(* CoDeSys 2.3.9.47 project: mqmod.pro *)
(* Libraries: C:\Program Files\WAGO Software\CoDeSys V2.3\Targets\WAGO\Libraries\32_Bit\oscat_basic_333.lib 9.2.16 18:15:54, WagoLibModbus_IP_01.lib 11.2.16 18:05:40, SysLibSockets.lib 22.5.14 16:16:32, WagoLibEthernet_01.lib 11.2.16 18:05:44, Standard.lib 20.5.14 08:13:26, Iecsfc.lib 16.5.13 14:00:50, SYSLIBCALLBACK.LIB 16.5.13 14:00:50 *)

(* PLC configuration (modules and I/O channels)
K-Bus [K_Bus] node 0, in %IB0 out %QB0 {KbusBusMode = 1; KbusCycleTime = 10000; KbusThreadPriority = 0; KbusSetOutputsToZeroOnApplicationStop = 1}
Modbus variables [PFC200MODBUS] node 1, in %IB0 out %QB0 {PlcStopBehaviour = 1; FiledbusErrorBehaviour = 1; TcpOperation = 1; TcpPort = 502; TcpTimeout = 600; UdpOperation = 1; UdpPort = 502; RtuOperation = 0; NodeId = 1; ResponseTimeout = 5000; Interface = 0; Baud = 115200; StopBits = 1; Parity = 1; FlowCtrl = 0; PhysInterface = 0}
Modbus-Master [MB_MASTER] node 2, in %IB0 out %QB0
*)

(* Global variable list: Globale_Variablen *)
VAR_GLOBAL
	xxSubscribe: BOOL := TRUE;
	xxPublish : BOOL     := TRUE;
	SubPubState : INT;
END_VAR

(* Data type *)
TYPE Buffer :
STRUCT
	data : ARRAY [0..MAX_RECEIVE_TCP_CLIENT] OF BYTE;
	iPos : DWORD := 0;
END_STRUCT
END_TYPE

(* Data type *)
TYPE ConnectFlags :
STRUCT
	xUsername     : BOOL;
	xPassword     : BOOL;
	xWillRetain   : BOOL;
	xWillQoS1     : BOOL;
    xWillQoS2     : BOOL;
	xWillFlag     : BOOL;
	xCleanSession : BOOL;
END_STRUCT
END_TYPE

(* Data type *)
TYPE FixedHeader :
STRUCT
	bMessageType : BYTE := 16#00;
	xDUP_FLAG    : BOOL := FALSE;
	xQos         : BYTE := 16#00; (*0,1,2*)
	xRetain      : BOOL := FALSE;
END_STRUCT
END_TYPE

(* Data type *)
TYPE FixedHeaderSub :
STRUCT
	bMessageType : BYTE := 8;
	xReserved         : BYTE := 2;
END_STRUCT
END_TYPE

(* Data type *)
TYPE Payload :
STRUCT
	data : ARRAY [0..30] OF BYTE;
	iPos : DWORD := 0;
END_STRUCT
END_TYPE

(* Data type *)
TYPE typReadReq :
STRUCT
	xReadRegister				:BOOL;
	wAdrBlockStart				:WORD;
	wAdrBlockQuantity			:WORD;
	ptDATA					:POINTER TO BYTE;
END_STRUCT
END_TYPE

(* Data type *)
TYPE typWriteReq
STRUCT
	xWriteRegister				:BOOL;
	wAdrBlockStart				:WORD;
	wAdrBlockQuantity			:WORD;
	ptDATA					:POINTER TO BYTE;
END_STRUCT
END_TYPE

(* POU PLC_PRG, ST *)
PROGRAM PLC_PRG
VAR

(*MQTT COMMUNICATION*)
	mqttClient: MQTT_CLIENT;
	xPublish: BOOL;
	xSubscribe: BOOL;
	socModbus : MODBUS_MASTER;

END_VAR
mqttClient(
xPublish := xxPublish, (* I/O variable to publish to a TOPIC *)
xSubscribe := xxSubscribe,  (* NOT SUPPORTED, but must be here for I/O *)
sIP:='10.210.10.29', (* IP of the MQTT Broker *)
wPortNumber:=1883,  (* PORT of the MQTT Broker *)
(* AUTH: When no authentication is needed, leave the following fields Blank *)
sUsername:='',  (* Username to connect with the MQTT Broker *)
sPassword:='' (* password to connect with the MQTT Broker *)
);

mqttClient.sTopic[1] 	:= 'si/upperstate'; 	(*40705 *)
mqttClient.sTopic[2] 	:= 'si/lowerstate';  	(*40707 *)
mqttClient.sTopic[3] 	:= 'si/activepower';	(*40149*)
mqttClient.sTopic[4]		:= 'si/activate';		(*40151*)
mqttClient.sTopic[5]		:= 'si/deactivate';	(*40151*)

mqttClient.sQoS := 16#00;
mqttClient.pTopic := 'soc';
mqttClient.pQoS := 16#00;
mqttClient.pRetained := FALSE;
mqttClient.pPayload :=  WORD_TO_STRING(socModbus.awRead[2]);(*STRING_TO_UDINT(g_SOC)*);

socModbus(
	xCONNECT:= TRUE,
	strIP_ADDRESS:= '10.210.10.63',
	wPORT:= 502,
	bUNIT_ID:= 16#03,
	bFUNCTION_CODE:= 16#03,
	wREAD_ADDRESS:= 30845 ,
	wREAD_QUANTITY:= 2 ,
 );
END_PROGRAM

(* POU MQTT/MQTT_CLIENT, ST *)
FUNCTION_BLOCK MQTT_CLIENT
VAR CONSTANT
	VERSION 	: BYTE := 16#03;
	Reserved   	: BYTE := 0;
	CONNECT     : BYTE := 1;
	CONNACK     : BYTE := 2;
	PUBLISH     : BYTE := 3;
	PUBACK      : BYTE := 4;
	PUBREC      : BYTE := 5;
	PUBREL      : BYTE := 6;
	PUBCOMP     : BYTE := 7;
	SUBSCRIBE   : BYTE := 8;
	SUBACK      : BYTE := 9;
	UNSUBSCRIBE : BYTE := 10;
	UNSUBACK    : BYTE := 11;
	PINGREQ     : BYTE := 12;
	PINGRESP    : BYTE := 13;
	DISCONNECT  : BYTE := 14;
	Reserved2   : BYTE := 15;

	CONNECTED   : INT := 30;
	NOT_CONNECTED: INT := 40;
	TIMEOUT : INT := 50;
	WAIT_RESPONSE : INT := 60;

	CONNECTION_TIMEOUT : TIME := t#10s;

	SUBSCRIBED : INT := 70;
	PUBLISHED : INT := 80;
	WAIT_RESPONSE_PUBLISH : INT := 90;
END_VAR

VAR
	fixedHeaderSub : BYTE;
	sendBuffer : Buffer;
	receiveBuffer : Buffer;
	fixedHeader: FixedHeader;
	variableHeader: Buffer;
	payLoad:  Buffer;
	connectFlags: ConnectFlags;
	tcpClient: TCP_Client;
	xTcpConnected: BOOL := FALSE;
	xStartSend: BOOL := FALSE;
	diReceiveCount: DINT;
	connectionTimer: TON;
	xTimeOut: BOOL;
	incomingMessageType: BYTE;
	eState: INT;
	xStartTimer: BOOL;

	rawdata : Buffer;
	b : Buffer;
	i :  DINT := 0;
	j:   DINT;
	x:  INT;
	z : INT := 0;

	c : BOOL; (*control state of subscription*)

	modControlValue : ARRAY[0..30] OF BYTE;
	RM : INT;
	LSB : INT;
	modValue : DINT;
	writeAdr : WORD;
	sstopic : ARRAY[0..20] OF BYTE;
	t : STRING;

	modbusMaster : MODBUS_MASTER;

END_VAR

VAR_INPUT
	sTopic: ARRAY[1..5] OF STRING;			(*SUB_TOPICS*)
	pTopic: STRING;						(*PUB_TOPICS*)
	pPayload: STRING;
	pRetained : BOOL;
	pQoS : BYTE;
	sQoS : BYTE;							(*von SMA ENERGY METER*)
	sIp : STRING;
	wPortNumber : WORD;
	sUsername : STRING;
	sPassword : STRING;
END_VAR

VAR_IN_OUT
	xPublish: BOOL;
	xSubscribe: BOOL;
END_VAR


VAR_OUTPUT
	xConnected : BOOL := FALSE;
	xBusy : BOOL := FALSE;
	activePowerVal : REAL;
END_VAR
tcpClient.sIPaddress := sIp;
tcpClient.wPortNumber := wPortNumber;

tcpClient.ptSendData := ADR(sendBuffer.data);
tcpClient.diSendCount := sendBuffer.iPos;

tcpClient(xOpenConnection:=TRUE,
xStartSend:=xStartSend,
aReceiveBuffer := receiveBuffer.data,
diReceiveCount := diReceiveCount);

xTcpConnected := tcpClient.xConnected;
xBusy := xStartSend;

IF NOT xTcpConnected THEN
	eState := NOT_CONNECTED;
	xConnected := FALSE;
 	RETURN;
END_IF;

(* INIT *)
payLoad.iPos := 0;
variableHeader.iPos := 0;

connectionTimer(IN:=xStartTimer, PT:=CONNECTION_TIMEOUT-t#2s);
xTimeOut := connectionTimer.Q;

(* Calculate the current state *)
IF xTimeOut THEN
	eState := TIMEOUT;
ELSIF eState <> CONNECTED AND eState <> TIMEOUT AND eState <> WAIT_RESPONSE THEN
	eState := NOT_CONNECTED;
END_IF

(* Execute current state *)
CASE eState OF

CONNECTED:
	IF diReceiveCount <> 0 THEN
		incomingMessageType := receiveBuffer.data[0];
		IF incomingMessageType = SHL(PINGRESP, 4) THEN
			xStartTimer := TRUE;
		END_IF
		IF incomingMessageType = SHL(PUBLISH, 4)  THEN
			_ARRAY_INIT(ADR(rawdata), SIZEOF(rawdata), 0);
			FOR i:=0 TO diReceiveCount-1 BY 1 DO
				rawdata.data[i] := receiveBuffer.data[i];
			END_FOR

			(*extract zuerst topic then payload*)
			RM := rawdata.data[1];
			LSB := rawdata.data[3];
			_ARRAY_INIT(ADR(sstopic), SIZEOF(sstopic), 0);
			i := 0; z := 0;
			FOR z := 4 TO LSB+3 DO
				sstopic[i]	:= rawdata.data[z];
				i := i + 1;
			END_FOR
			t := CONVERT_TO_STRING(sstopic);
			IF STRING_COMPARE(t, 'si/activepower') THEN
				writeAdr := 40149;
			ELSIF STRING_COMPARE(t, 'si/upperstate') THEN
				writeAdr := 40705;
			ELSIF STRING_COMPARE(t, 'si/lowerstate') THEN
				writeAdr := 40707;
			ELSIF STRING_COMPARE(t, 'si/activate') THEN
				writeAdr := 40151;
			ELSIF STRING_COMPARE(t, 'si/deactivate') THEN
				writeAdr := 40151;
			END_IF

			_ARRAY_INIT(ADR(modControlValue), SIZEOF(modControlValue), 0);
			i := 0; z := 0;
			FOR z := LSB+4 TO RM+1  DO
				modControlValue[i] := rawdata.data[z];
				i := i + 1;
			END_FOR
			modValue := REAL_TO_DINT(CONVERT_TO_REAL(modControlValue));
			z := 0;i := 0;
			modbusMaster(
				xCONNECT:= TRUE,
				strIP_ADDRESS:= '10.210.10.63',
				wPORT:= 502,
				bUNIT_ID:= 16#03,
				bFUNCTION_CODE:= 16#10,
				wWRITE_ADDRESS:= writeAdr, (*unterscheiden nach topic*)
				wWRITE_QUANTITY:= 2,
				value:= modValue);

			(*FOR z := 0 TO 15 BY 1 DO
				pValuesPrev[z] := pValues[z];
			END_FOR
			pValuePrev := CONVERT_TO_REAL(pValuesPrev);*)

			(*(*extract timestamp*)
			i := 0;
			FOR x := 13 TO 31 BY 1 DO
				IF x <> 17 AND x <> 20 AND x <> 23 AND x <> 26 AND x <> 29 THEN
						timestampPayload[i] := a.data[x];
					i := i + 1;
				END_IF
			END_FOR
			timestamp := EXTRACT_TIMESTAMP_FROM_PAYLOAD(timestampPayload);*)


		END_IF

		(*FURTHER QoS > 0*)
		IF incomingMessageType = SHL(PUBACK, 4)  THEN
			_ARRAY_INIT(ADR(b), SIZEOF(b), 0);
			FOR i:=0 TO diReceiveCount-1 BY 1 DO
				b.data[i] := receiveBuffer.data[i];
			END_FOR
		END_IF

		diReceiveCount := 0;
	END_IF

	c := xxPublish AND xxSubscribe;
	IF   c   THEN
		SubPubState := SUBSCRIBED;
	ELSE
		SubPubState := PUBLISHED;
	END_IF;

	CASE SubPubState OF
			SUBSCRIBED:
				IF xxSubscribe THEN
					_BUFFER_CLEAR(ADR(sendBuffer), SIZEOF(sendBuffer));

					fixedHeaderSub :=  BYTE_OF_BIT(FALSE, TRUE, FALSE, FALSE, FALSE, FALSE, FALSE, TRUE); (*FIXED_HEADER*)
					(*fixedHeaderSub.bMessageType := SUBSCRIBE;*)

					_BUFFER_PUSH(ADR(variableHeader), 16#00);(* Message ID *)
					_BUFFER_PUSH(ADR(variableHeader), 16#00);

					_BUFFER_PUSH_STRING(ADR(payLoad), sTopic[1] , TRUE);
					_BUFFER_PUSH(ADR(payLoad), sQoS); (*QoS 0 16#00*);

					(*Subscribe to multiple topics*)
					IF TRIM(sTopic[2]) <> ' ' THEN
						_BUFFER_PUSH_STRING(ADR(payLoad), sTopic[2] , TRUE);
						_BUFFER_PUSH(ADR(payLoad), sQoS); (*QoS 0 16#00*);
					END_IF
					IF TRIM(sTopic[3]) <> ' ' THEN
						_BUFFER_PUSH_STRING(ADR(payLoad), sTopic[3] , TRUE);
						_BUFFER_PUSH(ADR(payLoad), sQoS); (*QoS 0 16#00*);
					END_IF
					IF TRIM(sTopic[4]) <> ' ' THEN
						_BUFFER_PUSH_STRING(ADR(payLoad), sTopic[4] , TRUE);
						_BUFFER_PUSH(ADR(payLoad), sQoS); (*QoS 0 16#00*);
					END_IF
					IF TRIM(sTopic[5]) <> ' ' THEN
						_BUFFER_PUSH_STRING(ADR(payLoad), sTopic[4] , TRUE);
						_BUFFER_PUSH(ADR(payLoad), sQoS); (*QoS 0 16#00*);
					END_IF

					sendBuffer.iPos := 0;
					CREATE_MESSAGE_SUB(ADR(sendBuffer), fixedHeaderSub, variableHeader, payLoad);

					xxSubscribe := FALSE;
					(**xxSubscribe := TRUE;**)
					xStartSend := TRUE;
					SubPubState := PUBLISHED;
				END_IF

			 PUBLISHED:
				IF xxPublish THEN
					fixedHeader.bMessageType := PUBLISH;
					fixedHeader.xDUP_FLAG := FALSE;
					(*fixedHeader.xQos := 16#00; (* only QoS 0 supported *)*)
					fixedHeader.xQoS := pQoS;
					fixedHeader.xRetain := pRetained;

					_BUFFER_PUSH_STRING(ADR(variableHeader), pTopic, TRUE); (* Topic *)
					IF fixedHeader.xQos > 16#00 THEN
						_BUFFER_PUSH(ADR(variableHeader), 16#00);(* Message ID *)
						_BUFFER_PUSH(ADR(variableHeader), 16#00);
					END_IF

					_BUFFER_PUSH_STRING(ADR(payLoad), pPayload, FALSE);
					(*_BUFFER_PUSH(ADR(payLoad), sQoS); (*QoS 0 16#00*);*)

					sendBuffer.iPos := 0;
					CREATE_MESSAGE_PUB(ADR(sendBuffer), fixedHeader, variableHeader, payLoad);

					xxPublish := TRUE;
					xxSubscribe := TRUE;
					SubPubState := SUBSCRIBED;
					xStartSend := TRUE;
				END_IF
	END_CASE

NOT_CONNECTED:
	sendBuffer.iPos := 0;
	xStartTimer := FALSE;
	fixedHeader.bMessageType := CONNECT;

	_BUFFER_PUSH_STRING(ADR(variableHeader),'MQIsdp', TRUE); (* Protocol Name*)
	_BUFFER_PUSH(ADR(variableHeader), 3); (* Version Number*)

	connectFlags.xCleanSession := TRUE;
	connectFlags.xWillFlag     := FALSE;
	connectFlags.xWillQoS1     := FALSE;
	connectFlags.xWillQoS2     := FALSE;
	connectFlags.xWillRetain   := FALSE;
	IF LEN(sUsername) > 0 THEN
		connectFlags.xUsername := TRUE;
	ELSE
		connectFlags.xUsername := FALSE;
	END_IF
	IF LEN(sPassword) > 0 THEN
		connectFlags.xPassword := TRUE;
	ELSE
		connectFlags.xPassword := FALSE;
	END_IF

	_BUFFER_PUSH(ADR(variableHeader), BYTE_OF_BIT(FALSE,
															connectFlags.xCleanSession,
															connectFlags.xWillFlag,
															connectFlags.xWillQoS1,
															connectFlags.xWillQoS2,
															connectFlags.xWillRetain,
															connectFlags.xPassword,
															connectFlags.xUsername));

	_BUFFER_PUSH(ADR(variableHeader), 16#00);
	_BUFFER_PUSH(ADR(variableHeader), 16#0A); (* Keep Alive: 10s *)

	_BUFFER_PUSH_STRING(ADR(payload), 'PLC', TRUE); (* Client Identfier *)

	IF connectFlags.xUsername THEN
		_BUFFER_PUSH_STRING(ADR(payload), sUsername, TRUE); (* Username *)
	END_IF

	IF connectFlags.xPassword THEN
		_BUFFER_PUSH_STRING(ADR(payload), sPassword, TRUE); (* Password *)
	END_IF

	CREATE_MESSAGE(ADR(sendBuffer), fixedHeader, variableHeader, payLoad);

	eState := WAIT_RESPONSE;
	xStartSend := TRUE;

TIMEOUT:
	sendBuffer.iPos := 0;
	xStartTimer := FALSE;
	fixedHeader.bMessageType := PINGREQ;
	CREATE_MESSAGE(ADR(sendBuffer), fixedHeader, variableHeader, payLoad);

	eState := CONNECTED;
	xStartSend := TRUE;

WAIT_RESPONSE:
	incomingMessageType := receiveBuffer.data[0];
	IF incomingMessageType = SHL(CONNACK, 4) THEN
		(* TODO: Check return code *)
		xConnected := TRUE;
		xStartTimer := TRUE;
		eState := CONNECTED;
		diReceiveCount := 0;
	END_IF
END_CASE
END_FUNCTION_BLOCK

(* POU MODBUS/MODBUS_MASTER, ST *)
FUNCTION_BLOCK MODBUS_MASTER
VAR_INPUT

	xCONNECT						:BOOL:=TRUE;
	strIP_ADDRESS					:STRING;
	wPORT							:WORD := 502;	 (* Port-Nr.	*)
	bUNIT_ID							:BYTE := 16#03;
	bFUNCTION_CODE					:BYTE;
	wREAD_ADDRESS					:WORD;
	wREAD_QUANTITY					:WORD;
	ptREAD_DATA						:POINTER TO BYTE;
	wWRITE_ADDRESS				:WORD;
	wWRITE_QUANTITY				:WORD;
	value							: DINT;

END_VAR

VAR
	tTIME_OUT					:TIME:=t#15s;
	tCON_WATCHDOG				:TIME:=t#10s;
	xSEND						:BOOL;
	xIS_CONNECTED				:BOOL;
	wERROR						:WORD;
	bRESPONSE_UNIT_ID			:BYTE := 16#00;
	ptSEND_DATA						:POINTER TO BYTE;

	ETHERNET_MODBUSMASTER_TCP	:ETHERNET_MODBUSMASTER_TCP;

	awRead							:ARRAY[1..50] OF WORD;
	awWrite							:ARRAY[1..50] OF WORD;


	TON								:TON;

	xSEND_: BOOL;
	ton2: TON;
END_VAR

VAR_OUTPUT
END_VAR
awWrite[1]:=DWORD_TO_WORD(SHR(UDINT_TO_DWORD(value),16));
awWrite[2]:=UDINT_TO_WORD(value);



ETHERNET_MODBUSMASTER_TCP(
	xCONNECT:= xCONNECT,
	strIP_ADDRESS:= strIP_ADDRESS,
	wPORT:= 502,
	bUNIT_ID:= 3,
	bFUNCTION_CODE:= bFUNCTION_CODE,
	wREAD_ADDRESS:= wREAD_ADDRESS,
	wREAD_QUANTITY:=wREAD_QUANTITY ,
	ptREAD_DATA:= ADR(awRead),
	wWRITE_ADDRESS:= wWRITE_ADDRESS,
	wWRITE_QUANTITY:= wWRITE_QUANTITY,
	ptSEND_DATA:= ADR(awWrite),
	tTIME_OUT:= tTIME_OUT,
	tCON_WATCHDOG:= tCON_WATCHDOG,
	xSEND:=xSEND,
	xIS_CONNECTED=>xIS_CONNECTED,
	wERROR=>wERROR ,
	bRESPONSE_UNIT_ID=> bRESPONSE_UNIT_ID);

ton(in:=NOT ton2.q,
	pt:=t#5s);

ton2(in:=ton.q,
	pt:=t#5s);

IF ton2.Q THEN
	xSEND:=TRUE;
END_IF;
END_FUNCTION_BLOCK

(* POU Converters/CONVERT_TO_STRING, ST *)
FUNCTION CONVERT_TO_STRING : STRING
VAR_INPUT
	arTestArray: ARRAY[0..20] OF BYTE;
END_VAR
VAR
	pTestString: POINTER TO STRING;
	rRealValue: REAL;
END_VAR
pTestString:= ADR(arTestArray);

(*rRealValue:= STRING_TO_REAL(pTestString^);*)

CONVERT_TO_STRING := (pTestString^);
END_FUNCTION

(* POU Converters/CONVERT_TO_REAL, ST *)
FUNCTION CONVERT_TO_REAL : REAL
VAR_INPUT
	arTestArray: ARRAY[0..30] OF BYTE;
END_VAR
VAR
	pTestString: POINTER TO STRING;
	rRealValue: REAL;
END_VAR
pTestString:= ADR(arTestArray);

rRealValue:= STRING_TO_REAL(pTestString^);

CONVERT_TO_REAL := rRealValue;
END_FUNCTION

(* POU MQTT/MQTT_UTIL/_BUFFER_PUSH, ST *)
FUNCTION _BUFFER_PUSH : BOOL
VAR_INPUT
	PT  : POINTER TO Buffer;
	IN  : BYTE;
END_VAR

VAR
END_VAR
(* pushed data to a buffer array *)
PT^.data[PT^.iPos] := IN;

PT^.iPos := PT^.iPos + 1;

_BUFFER_PUSH := TRUE;
END_FUNCTION

(* POU MQTT/MQTT_UTIL/_BUFFER_PUSH_STRING, ST *)
FUNCTION _BUFFER_PUSH_STRING : BOOL
VAR_INPUT
	PT : POINTER TO Buffer;
	IN : STRING;
	INCLUDE_LENGTH : BOOL := FALSE;
END_VAR
VAR
	sPT : POINTER TO BYTE;
	iLen : DWORD;
	i : DWORD;
	nxtPtr: POINTER TO BYTE;
END_VAR
iLen := LEN(IN);
sPT := ADR(IN);

IF INCLUDE_LENGTH THEN
	_BUFFER_PUSH(PT, BYTE_OF_DWORD(iLen,1));
	_BUFFER_PUSH(PT, BYTE_OF_DWORD(iLen,0));
END_IF

FOR i:=0 TO iLen-1 BY 1 DO
	nxtPtr := sPT + i * SIZEOF(sPT^);
	_BUFFER_PUSH(PT, nxtPtr^);
END_FOR
END_FUNCTION

(* POU MQTT/MQTT_UTIL/CREATE_MESSAGE_SUB, ST *)
FUNCTION CREATE_MESSAGE_SUB : BOOL
VAR_INPUT
	PT          			:POINTER TO Buffer;
	fixedHeader      	: BYTE;
	variableHeader  	:Buffer;
	payLoad         		:Buffer;
END_VAR
VAR
	bTemp  			:BYTE;
	remainingLength	:DWORD;
END_VAR
(* FIXED HEADER *)
(* BYTE 1 *)
(*bTemp := bTemp OR SHL(fixedHeader, 4);*)
(*bTemp := bTemp OR fixedHeader;*)
bTemp := fixedHeader;

_BUFFER_PUSH(PT, bTemp);

(* BYTE 2 *)
remainingLength := variableHeader.iPos + payLoad.iPos;

ENCODE_REMAINING_LENGTH(PT, remainingLength);
(*_BUFFER_PUSH(PT, remainingLength);*)

(* VARIABLE HEADER *)
_BUFFER_CONCAT(PT, ADR(variableHeader));

(* PAYLOAD *)
_BUFFER_CONCAT(PT, ADR(payLoad));
END_FUNCTION

(* POU MQTT/MQTT_UTIL/ENCODE_REMAINING_LENGTH, ST *)
FUNCTION ENCODE_REMAINING_LENGTH : BOOL
VAR_INPUT
	PT : POINTER TO Buffer;
	LENGTH : DWORD;
END_VAR
VAR
	wPt : POINTER TO DWORD; (*4 bytes*)
	digit: DWORD;
	i: UINT;
END_VAR
wPt := ADR(LENGTH);

IF LENGTH = 0 THEN
	_BUFFER_PUSH(PT, 16#00);
	RETURN;
END_IF

WHILE LENGTH > 0 DO
	digit := LENGTH MOD 128;
	LENGTH := LENGTH / 128;
	
	IF LENGTH > 0 THEN
		digit := digit OR 16#80;
	END_IF
	_BUFFER_PUSH(PT, BYTE_OF_DWORD(digit,0));
END_WHILE
END_FUNCTION

(* POU MQTT/MQTT_UTIL/_BUFFER_CONCAT, ST *)
FUNCTION _BUFFER_CONCAT : BOOL
VAR_INPUT
	PT  : POINTER TO Buffer;
	PTContact  : POINTER TO Buffer;
END_VAR
VAR
	i: INT;
END_VAR
FOR i:=0 TO DWORD_TO_INT(PTContact^.iPos) -1 BY 1 DO
	_BUFFER_PUSH(PT, PTContact^.data[i]);
END_FOR
END_FUNCTION

(* POU MQTT/MQTT_UTIL/CREATE_MESSAGE_PUB, ST *)
FUNCTION CREATE_MESSAGE_PUB : BOOL
VAR_INPUT
	PT          : POINTER TO Buffer;
	fixedHeader     : FixedHeader;
	variableHeader  : Buffer;
	payLoad         : Buffer;
END_VAR
VAR
	bTemp  : BYTE;
	remainingLength: DWORD;
END_VAR
(* FIXED HEADER *)
(* BYTE 1 *)
bTemp := bTemp OR SHL(fixedHeader.bMessageType, 4) OR SHL(FixedHeader.xQos, 1);

BIT_LOAD_B(bTemp, FixedHeader.xDUP_FLAG, 3);
BIT_LOAD_B(bTemp, FixedHeader.xRetain, 0);

_BUFFER_PUSH(PT, bTemp);

(* BYTE 2 *)
remainingLength := variableHeader.iPos + payLoad.iPos;

ENCODE_REMAINING_LENGTH(PT, remainingLength);
(*_BUFFER_PUSH(PT, remainingLength);*)

(* VARIABLE HEADER *)
_BUFFER_CONCAT(PT, ADR(variableHeader));

(* PAYLOAD *)
_BUFFER_CONCAT(PT, ADR(payLoad));
END_FUNCTION

(* POU MQTT/MQTT_UTIL/CREATE_MESSAGE, ST *)
FUNCTION CREATE_MESSAGE : BOOL
VAR_INPUT
	PT          : POINTER TO Buffer;
	fixedHeader     : FixedHeader;
	variableHeader  : Buffer;
	payLoad         : Buffer;
END_VAR
VAR
	bTemp  : BYTE;
	remainingLength: DWORD;
END_VAR
(* FIXED HEADER *)
(* BYTE 1 *)
bTemp := bTemp OR SHL(fixedHeader.bMessageType, 4) OR SHL(FixedHeader.xQos, 1);

BIT_LOAD_B(bTemp, FixedHeader.xDUP_FLAG, 3);
BIT_LOAD_B(bTemp, FixedHeader.xRetain, 0);

_BUFFER_PUSH(PT, bTemp);

(* BYTE 2 *)
remainingLength := variableHeader.iPos + payLoad.iPos;

ENCODE_REMAINING_LENGTH(PT, remainingLength);
(*_BUFFER_PUSH(PT, remainingLength);*)

(* VARIABLE HEADER *)
_BUFFER_CONCAT(PT, ADR(variableHeader));

(* PAYLOAD *)
_BUFFER_CONCAT(PT, ADR(payLoad));
END_FUNCTION

(* POU MQTT/MQTT_UTIL/_BUFFER_SET, ST *)
FUNCTION _BUFFER_SET : BOOL
VAR_INPUT
	PT  : POINTER TO Buffer;
	IN  : BYTE;
	POS : UINT := 0;
END_VAR
VAR
END_VAR
PT^.data[POS] := IN;

IF PT^.iPos < POS THEN
	PT^.iPos := POS;
END_IF
END_FUNCTION

(* POU MQTT/MQTT_UTIL/_PAYLOAD_PUSH, ST *)
FUNCTION _PAYLOAD_PUSH : BOOL
VAR_INPUT
	PT  : POINTER TO Payload;
	IN  : BYTE;
END_VAR
VAR
END_VAR
(* pushed data to a buffer array *)
PT^.data[PT^.iPos] := IN;

PT^.iPos := PT^.iPos + 1;

_PAYLOAD_PUSH := TRUE;
END_FUNCTION

(* POU MQTT/MQTT_UTIL/EXTRACT_TIMESTAMP_FROM_PAYLOAD, ST *)
FUNCTION EXTRACT_TIMESTAMP_FROM_PAYLOAD : DATE_AND_TIME
VAR_INPUT
	data: ARRAY[0..13] OF BYTE;
END_VAR
VAR
	pTestString: POINTER TO STRING;
	pTestStringA: ARRAY[0..5] OF POINTER TO STRING;
	timestamp: DATE_AND_TIME;
	i: INT := 0;
	j : INT := 0;
	yeara : ARRAY[0..4] OF BYTE;
	montha : ARRAY[0..2] OF BYTE;
	daya : ARRAY[0..2] OF BYTE;
	houra : ARRAY[0..2] OF BYTE;
	minutea : ARRAY[0..2] OF BYTE;
	seconda : ARRAY[0..2] OF BYTE;

	year1: INT;
	month1: INT;
	day1: INT;
	hour1: INT;
	minute1:INT;
	second1:INT;

	rRealValue: BOOL;
END_VAR
FOR i := 0 TO 13 BY 1 DO
	IF i <= 3				 		THEN yeara[i] := data[i];
	ELSIF  i > 3 AND i <= 5 			THEN IF j > 1 THEN j := 0;  END_IF; 		montha[j] := data[i];  	 j:=j+1;
	ELSIF  i > 5 AND i <= 7 			THEN IF j > 1 THEN j := 0;  END_IF;  	daya[j] := data[i]; 	 j:=j+1;
	ELSIF  i >= 8 AND i <= 9 			THEN IF j > 1 THEN j := 0;  END_IF; 		houra[j] := data[i];   	 j:=j+1;
	ELSIF  i > 9 AND i <= 11 			THEN IF j > 1 THEN j := 0;  END_IF; 		minutea[j] := data[i];   j:=j+1;
	ELSIF  i > 11 AND i <= 13 		THEN IF j > 1 THEN j := 0;   END_IF;  	seconda[j] := data[i];  j:=j+1;
	END_IF;
END_FOR

(*pTestString:= ADR(yeara);
iValue:= STRING_TO_INT(pTestString^);
EXTRACT_TIMESTAMP_FROM_PAYLOAD := iValue;*)

pTestStringA[0] := ADR(yeara);
pTestStringA[1] := ADR(montha);
pTestStringA[2] := ADR(daya);
pTestStringA[3] := ADR(houra);
pTestStringA[4] := ADR(minutea);
pTestStringA[5] := ADR(seconda);

(*pTestString	 :=      ADR(yeara);
year1		 :=  	STRING_TO_INT(pTestString^);
EXTRACT_TIMESTAMP_FROM_PAYLOAD := year1;*)

year1:=  		STRING_TO_INT(pTestStringA[0]^);
month1 :=  	STRING_TO_INT(pTestStringA[1]^);
day1 := 		STRING_TO_INT(pTestStringA[2]^);
hour1 := 		STRING_TO_INT(pTestStringA[3]^);
minute1 := 	STRING_TO_INT(pTestStringA[4]^);
second1 :=  	STRING_TO_INT(pTestStringA[5]^);


EXTRACT_TIMESTAMP_FROM_PAYLOAD := SET_DT(
	year := year1,
	month := month1,
	day := day1  ,
	HOUR := hour1,
	MINUTE := minute1,
	SECOND := second1);
END_FUNCTION
